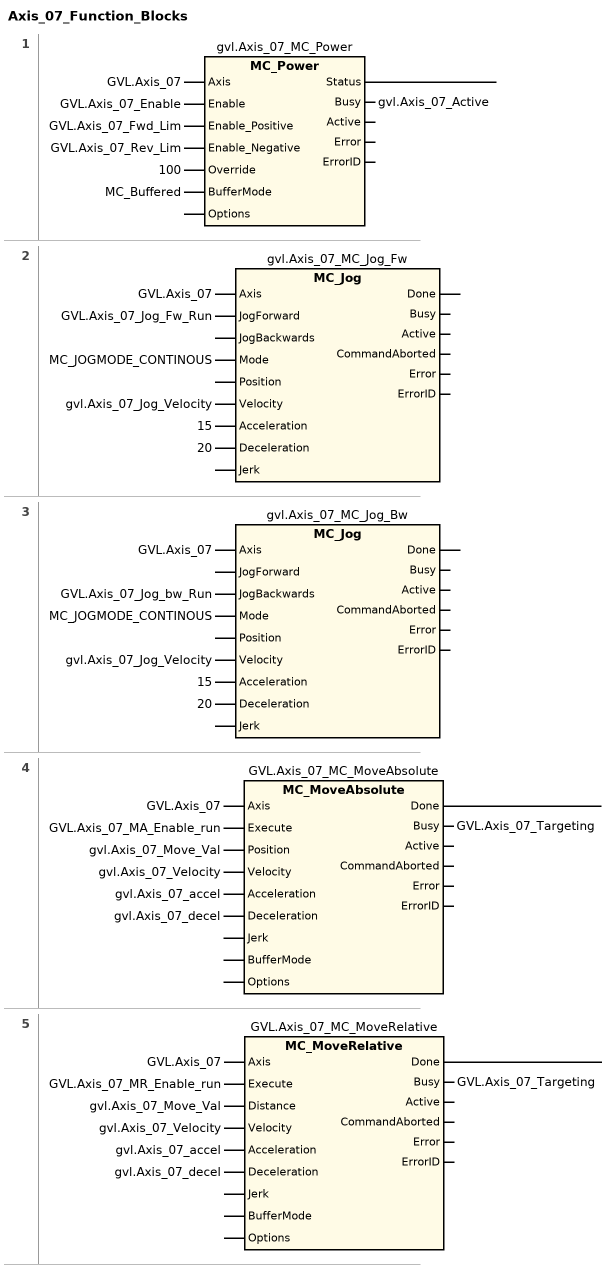
// NETWORK 1
gvl.Axis_07_MC_Power(
    Axis := GVL.Axis_07,
    Enable := GVL.Axis_07_Enable,
    Enable_Positive := GVL.Axis_07_Fwd_Lim,
    Enable_Negative := GVL.Axis_07_Rev_Lim,
    Override := 100,
    BufferMode := MC_Buffered,
    Busy => gvl.Axis_07_Active); // MC_Power

// NETWORK 2
gvl.Axis_07_MC_Jog_Fw(
    Axis := GVL.Axis_07,
    JogForward := GVL.Axis_07_Jog_Fw_Run,
    Mode := MC_JOGMODE_CONTINOUS,
    Velocity := gvl.Axis_07_Jog_Velocity,
    Acceleration := 15,
    Deceleration := 20); // MC_Jog

// NETWORK 3
gvl.Axis_07_MC_Jog_Bw(
    Axis := GVL.Axis_07,
    JogBackwards := GVL.Axis_07_Jog_bw_Run,
    Mode := MC_JOGMODE_CONTINOUS,
    Velocity := gvl.Axis_07_Jog_Velocity,
    Acceleration := 15,
    Deceleration := 20); // MC_Jog

// NETWORK 4
GVL.Axis_07_MC_MoveAbsolute(
    Axis := GVL.Axis_07,
    Execute := GVL.Axis_07_MA_Enable_run,
    Position := gvl.Axis_07_Move_Val,
    Velocity := gvl.Axis_07_Velocity,
    Acceleration := gvl.Axis_07_accel,
    Deceleration := gvl.Axis_07_decel,
    Busy => GVL.Axis_07_Targeting); // MC_MoveAbsolute

// NETWORK 5
GVL.Axis_07_MC_MoveRelative(
    Axis := GVL.Axis_07,
    Execute := GVL.Axis_07_MR_Enable_run,
    Distance := gvl.Axis_07_Move_Val,
    Velocity := gvl.Axis_07_Velocity,
    Acceleration := gvl.Axis_07_accel,
    Deceleration := gvl.Axis_07_decel,
    Busy => GVL.Axis_07_Targeting); // MC_MoveRelative

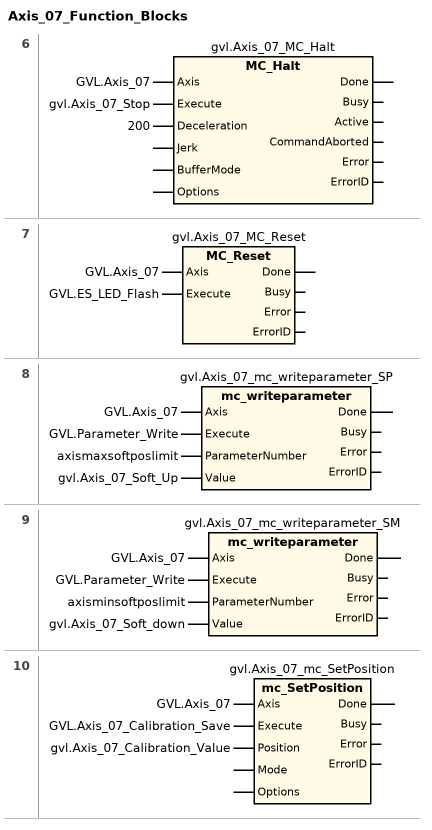
// NETWORK 6
gvl.Axis_07_MC_Halt(Axis := GVL.Axis_07, Execute := gvl.Axis_07_Stop, Deceleration := 200); // MC_Halt

// NETWORK 7
gvl.Axis_07_MC_Reset(Axis := GVL.Axis_07, Execute := GVL.ES_LED_Flash); // MC_Reset

// NETWORK 8
gvl.Axis_07_mc_writeparameter_SP(
    Axis := GVL.Axis_07,
    Execute := GVL.Parameter_Write,
    ParameterNumber := axismaxsoftposlimit,
    Value := gvl.Axis_07_Soft_Up); // mc_writeparameter

// NETWORK 9
gvl.Axis_07_mc_writeparameter_SM(
    Axis := GVL.Axis_07,
    Execute := GVL.Parameter_Write,
    ParameterNumber := axisminsoftposlimit,
    Value := gvl.Axis_07_Soft_down); // mc_writeparameter

// NETWORK 10
gvl.Axis_07_mc_SetPosition(
    Axis := GVL.Axis_07,
    Execute := GVL.Axis_07_Calibration_Save,
    Position := gvl.Axis_07_Calibration_Value); // mc_SetPosition

END_PROGRAM

// ---- POUs/Axis_07_Logic.TcPOU
PROGRAM Axis_07_Logic
VAR
	TON_0: TON;
	TON_1: TON;
	TON_2: TON;
	TON_3: TON;
	Axis_07_Velocity_Range: LREAL;
	Axis_07_Velocity_Scale: LREAL;
	Axis_07_Velocity_Raw: LREAL;
	Axis_07_Soft_Range: LREAL;
	Axis_07_Soft_Position: LREAL;
	Axis_07_Soft_Position_In_Range: LREAL;
END_VAR

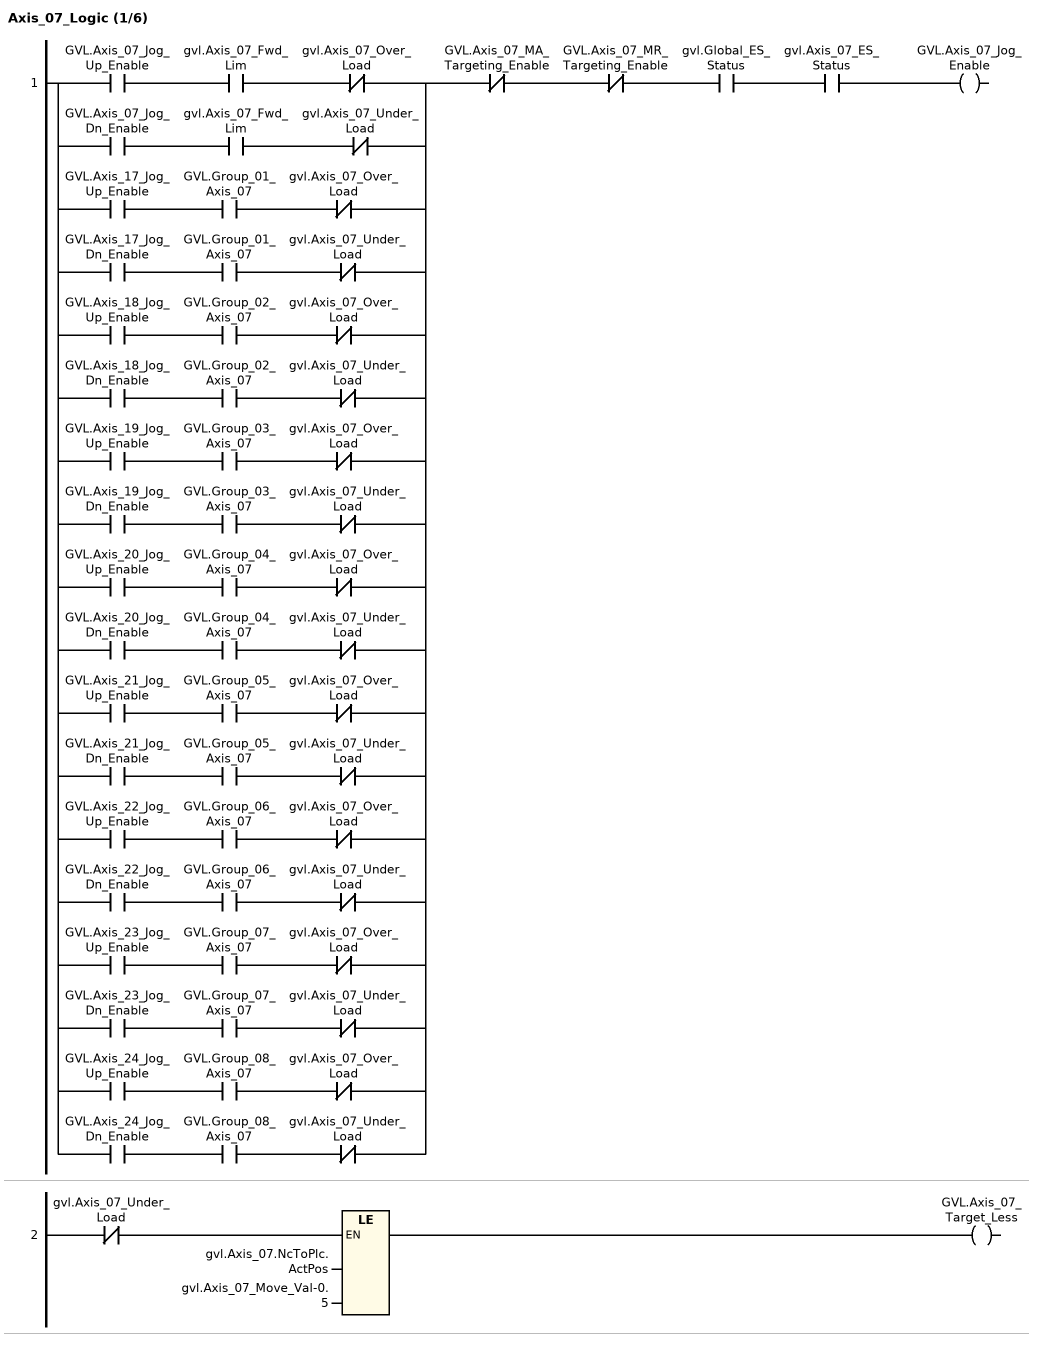
// NETWORK 1
GVL.Axis_07_Jog_Enable := (GVL.Axis_07_Jog_Up_Enable AND gvl.Axis_07_Fwd_Lim AND NOT gvl.Axis_07_Over_Load OR GVL.Axis_07_Jog_Dn_Enable AND gvl.Axis_07_Fwd_Lim AND NOT gvl.Axis_07_Under_Load OR GVL.Axis_17_Jog_Up_Enable AND GVL.Group_01_Axis_07 AND NOT gvl.Axis_07_Over_Load OR GVL.Axis_17_Jog_Dn_Enable AND GVL.Group_01_Axis_07 AND NOT gvl.Axis_07_Under_Load OR GVL.Axis_18_Jog_Up_Enable AND GVL.Group_02_Axis_07 AND NOT gvl.Axis_07_Over_Load OR GVL.Axis_18_Jog_Dn_Enable AND GVL.Group_02_Axis_07 AND NOT gvl.Axis_07_Under_Load OR GVL.Axis_19_Jog_Up_Enable AND GVL.Group_03_Axis_07 AND NOT gvl.Axis_07_Over_Load OR GVL.Axis_19_Jog_Dn_Enable AND GVL.Group_03_Axis_07 AND NOT gvl.Axis_07_Under_Load OR GVL.Axis_20_Jog_Up_Enable AND GVL.Group_04_Axis_07 AND NOT gvl.Axis_07_Over_Load OR GVL.Axis_20_Jog_Dn_Enable AND GVL.Group_04_Axis_07 AND NOT gvl.Axis_07_Under_Load OR GVL.Axis_21_Jog_Up_Enable AND GVL.Group_05_Axis_07 AND NOT gvl.Axis_07_Over_Load OR GVL.Axis_21_Jog_Dn_Enable AND GVL.Group_05_Axis_07 AND NOT gvl.Axis_07_Under_Load OR GVL.Axis_22_Jog_Up_Enable AND GVL.Group_06_Axis_07 AND NOT gvl.Axis_07_Over_Load OR GVL.Axis_22_Jog_Dn_Enable AND GVL.Group_06_Axis_07 AND NOT gvl.Axis_07_Under_Load OR GVL.Axis_23_Jog_Up_Enable AND GVL.Group_07_Axis_07 AND NOT gvl.Axis_07_Over_Load OR GVL.Axis_23_Jog_Dn_Enable AND GVL.Group_07_Axis_07 AND NOT gvl.Axis_07_Under_Load OR GVL.Axis_24_Jog_Up_Enable AND GVL.Group_08_Axis_07 AND NOT gvl.Axis_07_Over_Load OR GVL.Axis_24_Jog_Dn_Enable AND GVL.Group_08_Axis_07 AND NOT gvl.Axis_07_Under_Load) AND NOT GVL.Axis_07_MA_Targeting_Enable AND NOT GVL.Axis_07_MR_Targeting_Enable AND gvl.Global_ES_Status AND gvl.Axis_07_ES_Status;

// NETWORK 2
GVL.Axis_07_Target_Less := NOT gvl.Axis_07_Under_Load AND gvl.Axis_07.NcToPlc.ActPos <= (gvl.Axis_07_Move_Val-0.5);

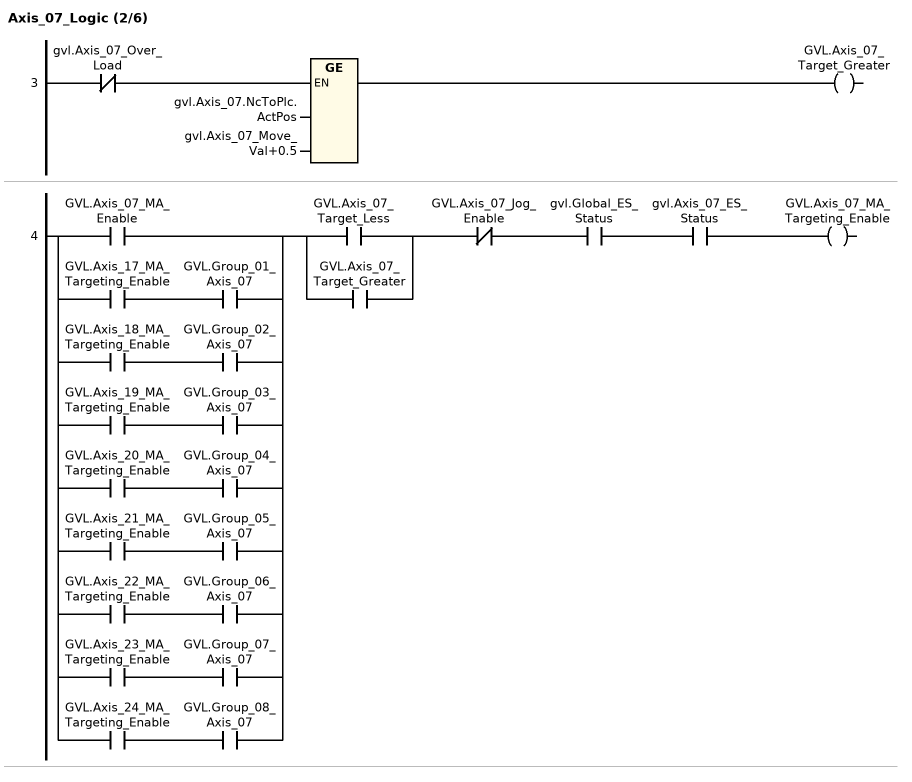
// NETWORK 3
GVL.Axis_07_Target_Greater := NOT gvl.Axis_07_Over_Load AND gvl.Axis_07.NcToPlc.ActPos >= (gvl.Axis_07_Move_Val+0.5);

// NETWORK 4
GVL.Axis_07_MA_Targeting_Enable := (GVL.Axis_07_MA_Enable OR GVL.Axis_17_MA_Targeting_Enable AND GVL.Group_01_Axis_07 OR GVL.Axis_18_MA_Targeting_Enable AND GVL.Group_02_Axis_07 OR GVL.Axis_19_MA_Targeting_Enable AND GVL.Group_03_Axis_07 OR GVL.Axis_20_MA_Targeting_Enable AND GVL.Group_04_Axis_07 OR GVL.Axis_21_MA_Targeting_Enable AND GVL.Group_05_Axis_07 OR GVL.Axis_22_MA_Targeting_Enable AND GVL.Group_06_Axis_07 OR GVL.Axis_23_MA_Targeting_Enable AND GVL.Group_07_Axis_07 OR GVL.Axis_24_MA_Targeting_Enable AND GVL.Group_08_Axis_07) AND (GVL.Axis_07_Target_Less OR GVL.Axis_07_Target_Greater) AND NOT GVL.Axis_07_Jog_Enable AND gvl.Global_ES_Status AND gvl.Axis_07_ES_Status;

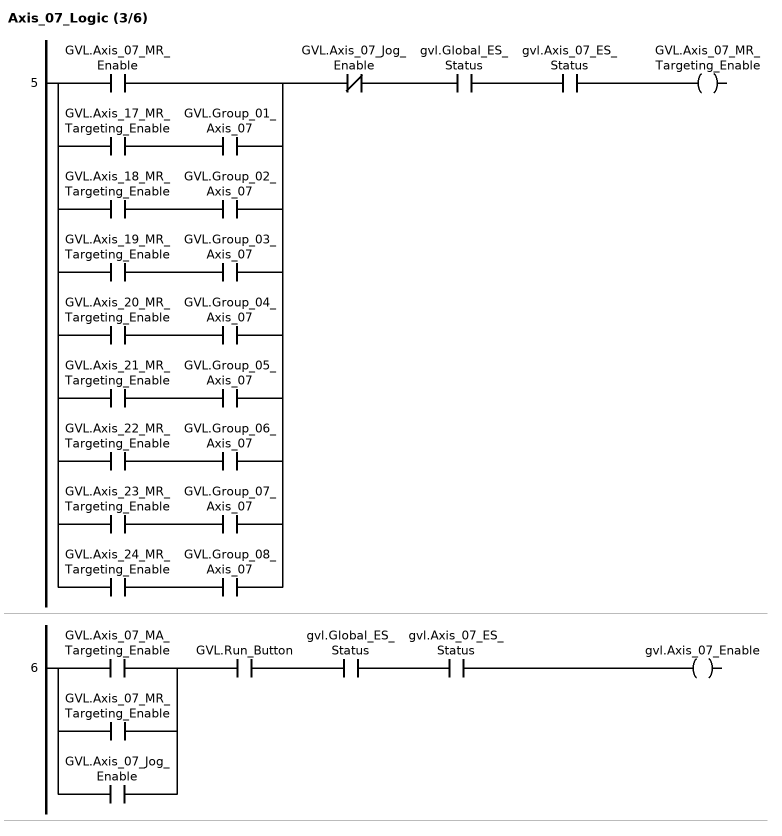
// NETWORK 5
GVL.Axis_07_MR_Targeting_Enable := (GVL.Axis_07_MR_Enable OR GVL.Axis_17_MR_Targeting_Enable AND GVL.Group_01_Axis_07 OR GVL.Axis_18_MR_Targeting_Enable AND GVL.Group_02_Axis_07 OR GVL.Axis_19_MR_Targeting_Enable AND GVL.Group_03_Axis_07 OR GVL.Axis_20_MR_Targeting_Enable AND GVL.Group_04_Axis_07 OR GVL.Axis_21_MR_Targeting_Enable AND GVL.Group_05_Axis_07 OR GVL.Axis_22_MR_Targeting_Enable AND GVL.Group_06_Axis_07 OR GVL.Axis_23_MR_Targeting_Enable AND GVL.Group_07_Axis_07 OR GVL.Axis_24_MR_Targeting_Enable AND GVL.Group_08_Axis_07) AND NOT GVL.Axis_07_Jog_Enable AND gvl.Global_ES_Status AND gvl.Axis_07_ES_Status;

// NETWORK 6
gvl.Axis_07_Enable := (GVL.Axis_07_MA_Targeting_Enable OR GVL.Axis_07_MR_Targeting_Enable OR GVL.Axis_07_Jog_Enable) AND GVL.Run_Button AND gvl.Global_ES_Status AND gvl.Axis_07_ES_Status;

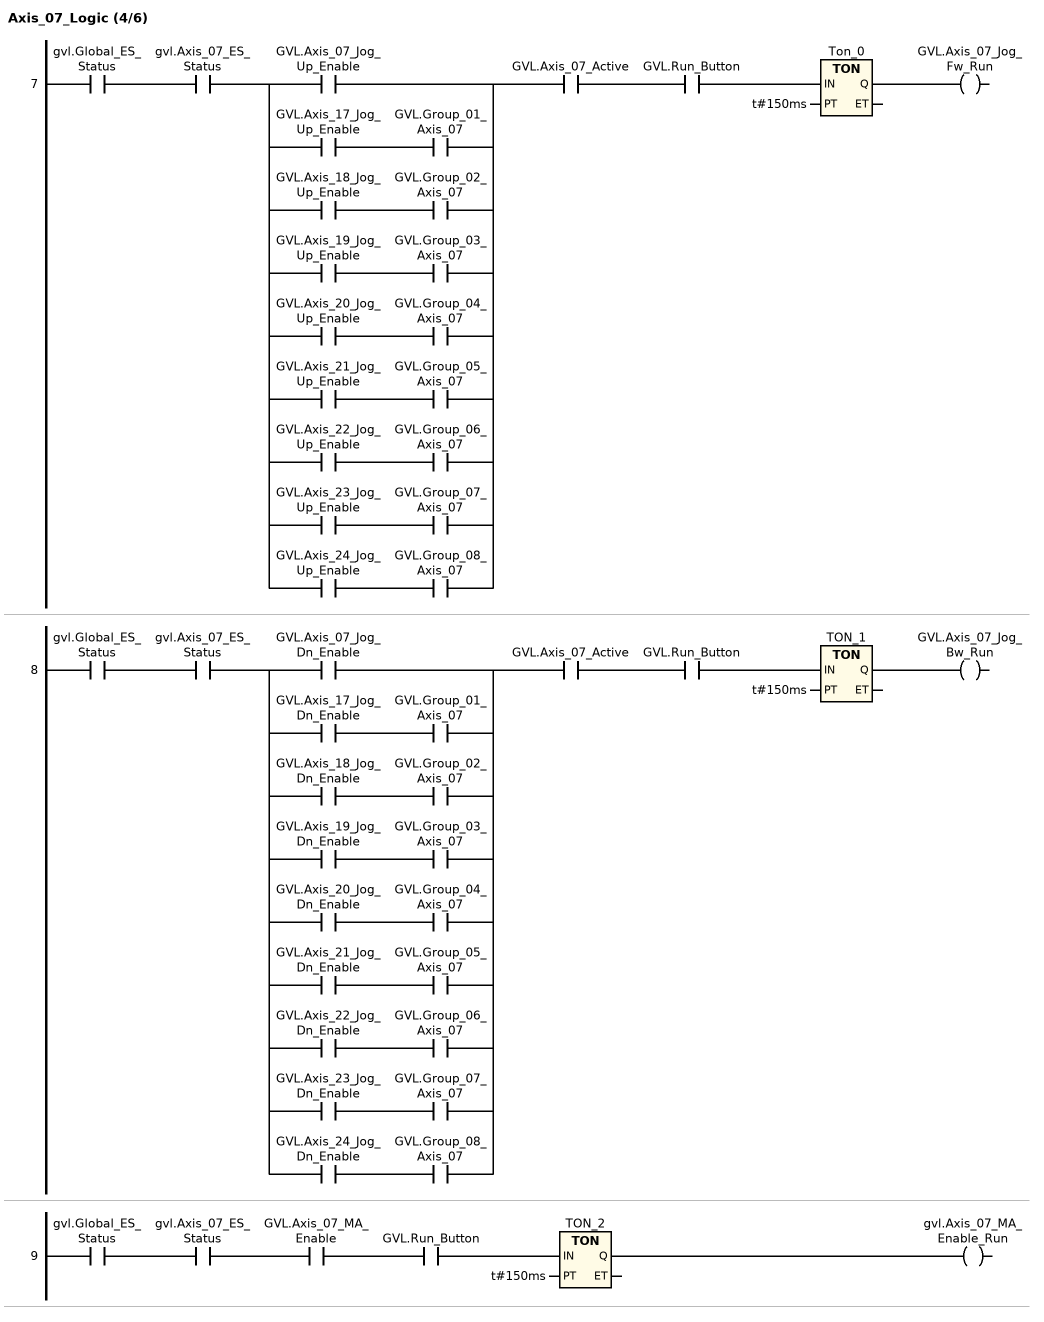
// NETWORK 7
Ton_0(IN := gvl.Global_ES_Status AND gvl.Axis_07_ES_Status AND (GVL.Axis_07_Jog_Up_Enable OR GVL.Axis_17_Jog_Up_Enable AND GVL.Group_01_Axis_07 OR GVL.Axis_18_Jog_Up_Enable AND GVL.Group_02_Axis_07 OR GVL.Axis_19_Jog_Up_Enable AND GVL.Group_03_Axis_07 OR GVL.Axis_20_Jog_Up_Enable AND GVL.Group_04_Axis_07 OR GVL.Axis_21_Jog_Up_Enable AND GVL.Group_05_Axis_07 OR GVL.Axis_22_Jog_Up_Enable AND GVL.Group_06_Axis_07 OR GVL.Axis_23_Jog_Up_Enable AND GVL.Group_07_Axis_07 OR GVL.Axis_24_Jog_Up_Enable AND GVL.Group_08_Axis_07) AND GVL.Axis_07_Active AND GVL.Run_Button, PT := t#150ms); // TON
GVL.Axis_07_Jog_Fw_Run := Ton_0.Q;

// NETWORK 8
TON_1(IN := gvl.Global_ES_Status AND gvl.Axis_07_ES_Status AND (GVL.Axis_07_Jog_Dn_Enable OR GVL.Axis_17_Jog_Dn_Enable AND GVL.Group_01_Axis_07 OR GVL.Axis_18_Jog_Dn_Enable AND GVL.Group_02_Axis_07 OR GVL.Axis_19_Jog_Dn_Enable AND GVL.Group_03_Axis_07 OR GVL.Axis_20_Jog_Dn_Enable AND GVL.Group_04_Axis_07 OR GVL.Axis_21_Jog_Dn_Enable AND GVL.Group_05_Axis_07 OR GVL.Axis_22_Jog_Dn_Enable AND GVL.Group_06_Axis_07 OR GVL.Axis_23_Jog_Dn_Enable AND GVL.Group_07_Axis_07 OR GVL.Axis_24_Jog_Dn_Enable AND GVL.Group_08_Axis_07) AND GVL.Axis_07_Active AND GVL.Run_Button, PT := t#150ms); // TON
GVL.Axis_07_Jog_Bw_Run := TON_1.Q;

// NETWORK 9
TON_2(IN := gvl.Global_ES_Status AND gvl.Axis_07_ES_Status AND GVL.Axis_07_MA_Enable AND GVL.Run_Button, PT := t#150ms); // TON
gvl.Axis_07_MA_Enable_Run := TON_2.Q;

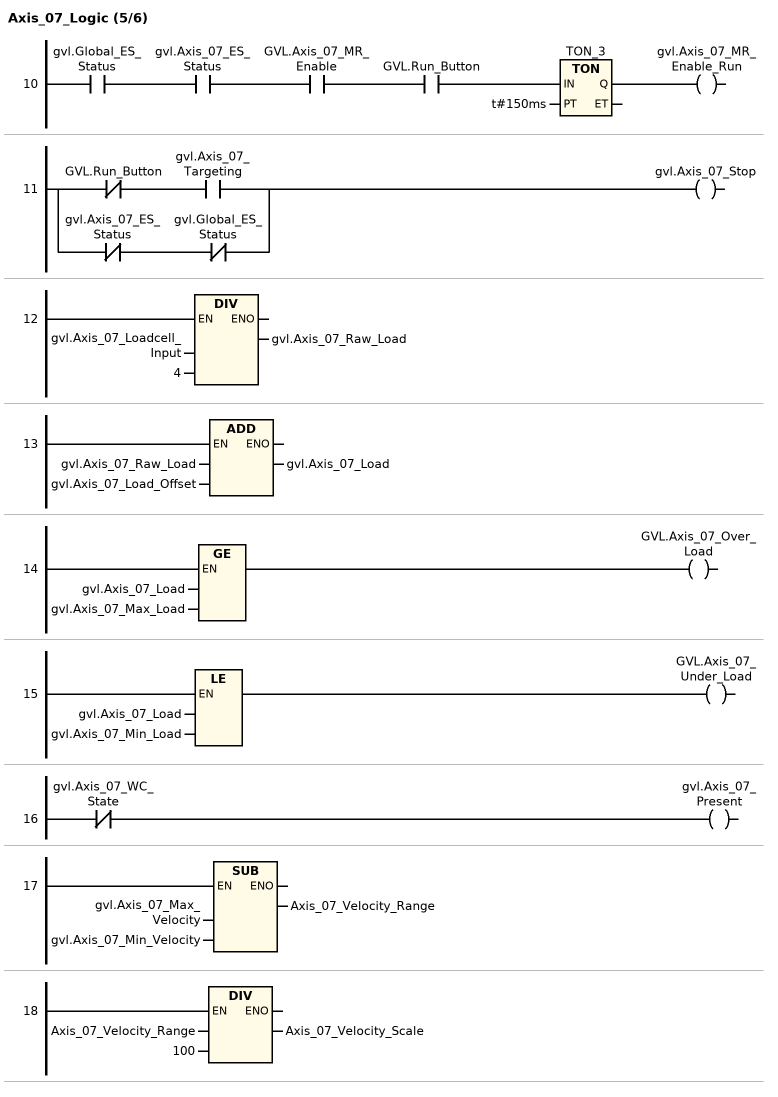
// NETWORK 10
TON_3(IN := gvl.Global_ES_Status AND gvl.Axis_07_ES_Status AND GVL.Axis_07_MR_Enable AND GVL.Run_Button, PT := t#150ms); // TON
gvl.Axis_07_MR_Enable_Run := TON_3.Q;

// NETWORK 11
gvl.Axis_07_Stop := NOT GVL.Run_Button AND gvl.Axis_07_Targeting OR NOT gvl.Axis_07_ES_Status AND NOT gvl.Global_ES_Status;

// NETWORK 12
gvl.Axis_07_Raw_Load := gvl.Axis_07_Loadcell_Input / 4;

// NETWORK 13
gvl.Axis_07_Load := gvl.Axis_07_Raw_Load + gvl.Axis_07_Load_Offset;

// NETWORK 14
GVL.Axis_07_Over_Load := gvl.Axis_07_Load >= gvl.Axis_07_Max_Load;

// NETWORK 15
GVL.Axis_07_Under_Load := gvl.Axis_07_Load <= gvl.Axis_07_Min_Load;

// NETWORK 16
gvl.Axis_07_Present := NOT gvl.Axis_07_WC_State;

// NETWORK 17
Axis_07_Velocity_Range := gvl.Axis_07_Max_Velocity - gvl.Axis_07_Min_Velocity;

// NETWORK 18
Axis_07_Velocity_Scale := Axis_07_Velocity_Range / 100;

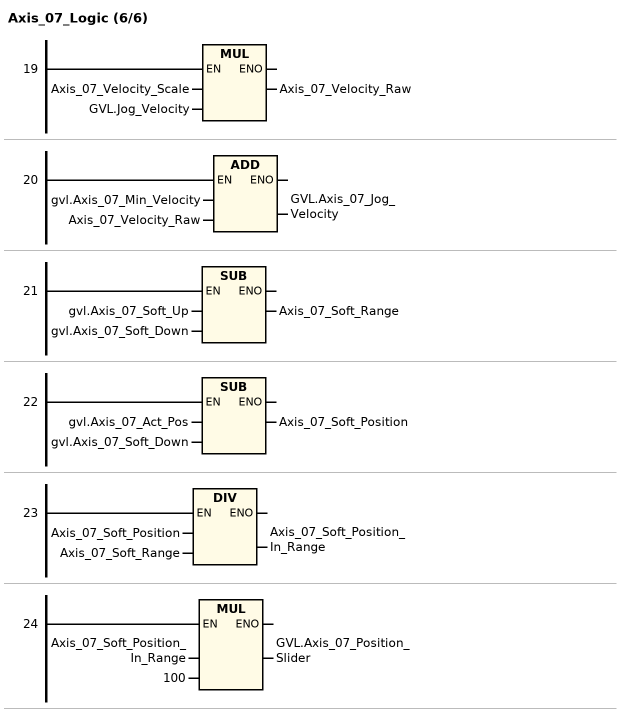
// NETWORK 19
Axis_07_Velocity_Raw := Axis_07_Velocity_Scale * GVL.Jog_Velocity;

// NETWORK 20
GVL.Axis_07_Jog_Velocity := gvl.Axis_07_Min_Velocity + Axis_07_Velocity_Raw;

// NETWORK 21
Axis_07_Soft_Range := gvl.Axis_07_Soft_Up - gvl.Axis_07_Soft_Down;

// NETWORK 22
Axis_07_Soft_Position := gvl.Axis_07_Act_Pos - gvl.Axis_07_Soft_Down;

// NETWORK 23
Axis_07_Soft_Position_In_Range := Axis_07_Soft_Position / Axis_07_Soft_Range;

// NETWORK 24
GVL.Axis_07_Position_Slider := Axis_07_Soft_Position_In_Range * 100;

END_PROGRAM

// ---- POUs/Axis_08_Function_Blocks.TcPOU
PROGRAM Axis_08_Function_Blocks
VAR
END_VAR

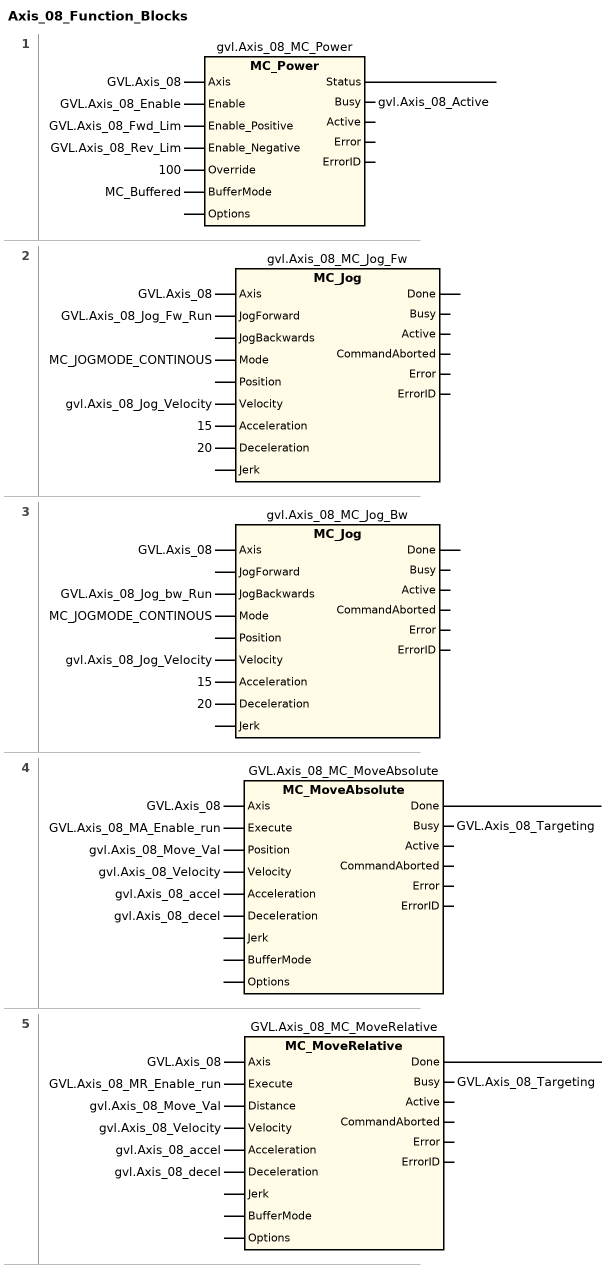
// NETWORK 1
gvl.Axis_08_MC_Power(
    Axis := GVL.Axis_08,
    Enable := GVL.Axis_08_Enable,
    Enable_Positive := GVL.Axis_08_Fwd_Lim,
    Enable_Negative := GVL.Axis_08_Rev_Lim,
    Override := 100,
    BufferMode := MC_Buffered,
    Busy => gvl.Axis_08_Active); // MC_Power

// NETWORK 2
gvl.Axis_08_MC_Jog_Fw(
    Axis := GVL.Axis_08,
    JogForward := GVL.Axis_08_Jog_Fw_Run,
    Mode := MC_JOGMODE_CONTINOUS,
    Velocity := gvl.Axis_08_Jog_Velocity,
    Acceleration := 15,
    Deceleration := 20); // MC_Jog

// NETWORK 3
gvl.Axis_08_MC_Jog_Bw(
    Axis := GVL.Axis_08,
    JogBackwards := GVL.Axis_08_Jog_bw_Run,
    Mode := MC_JOGMODE_CONTINOUS,
    Velocity := gvl.Axis_08_Jog_Velocity,
    Acceleration := 15,
    Deceleration := 20); // MC_Jog

// NETWORK 4
GVL.Axis_08_MC_MoveAbsolute(
    Axis := GVL.Axis_08,
    Execute := GVL.Axis_08_MA_Enable_run,
    Position := gvl.Axis_08_Move_Val,
    Velocity := gvl.Axis_08_Velocity,
    Acceleration := gvl.Axis_08_accel,
    Deceleration := gvl.Axis_08_decel,
    Busy => GVL.Axis_08_Targeting); // MC_MoveAbsolute

// NETWORK 5
GVL.Axis_08_MC_MoveRelative(
    Axis := GVL.Axis_08,
    Execute := GVL.Axis_08_MR_Enable_run,
    Distance := gvl.Axis_08_Move_Val,
    Velocity := gvl.Axis_08_Velocity,
    Acceleration := gvl.Axis_08_accel,
    Deceleration := gvl.Axis_08_decel,
    Busy => GVL.Axis_08_Targeting); // MC_MoveRelative

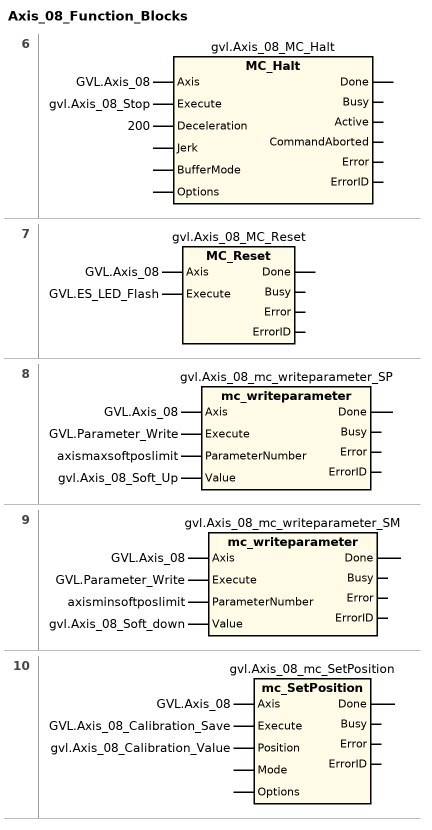
// NETWORK 6
gvl.Axis_08_MC_Halt(Axis := GVL.Axis_08, Execute := gvl.Axis_08_Stop, Deceleration := 200); // MC_Halt

// NETWORK 7
gvl.Axis_08_MC_Reset(Axis := GVL.Axis_08, Execute := GVL.ES_LED_Flash); // MC_Reset

// NETWORK 8
gvl.Axis_08_mc_writeparameter_SP(
    Axis := GVL.Axis_08,
    Execute := GVL.Parameter_Write,
    ParameterNumber := axismaxsoftposlimit,
    Value := gvl.Axis_08_Soft_Up); // mc_writeparameter

// NETWORK 9
gvl.Axis_08_mc_writeparameter_SM(
    Axis := GVL.Axis_08,
    Execute := GVL.Parameter_Write,
    ParameterNumber := axisminsoftposlimit,
    Value := gvl.Axis_08_Soft_down); // mc_writeparameter

// NETWORK 10
gvl.Axis_08_mc_SetPosition(
    Axis := GVL.Axis_08,
    Execute := GVL.Axis_08_Calibration_Save,
    Position := gvl.Axis_08_Calibration_Value); // mc_SetPosition

END_PROGRAM

// ---- POUs/Axis_08_Logic.TcPOU
PROGRAM Axis_08_Logic
VAR
	TON_0: TON;
	TON_1: TON;
	TON_2: TON;
	TON_3: TON;
	Axis_08_Velocity_Range: LREAL;
	Axis_08_Velocity_Scale: LREAL;
	Axis_08_Velocity_Raw: LREAL;
	Axis_08_Soft_Range: LREAL;
	Axis_08_Soft_Position: LREAL;
	Axis_08_Soft_Position_In_Range: LREAL;
END_VAR

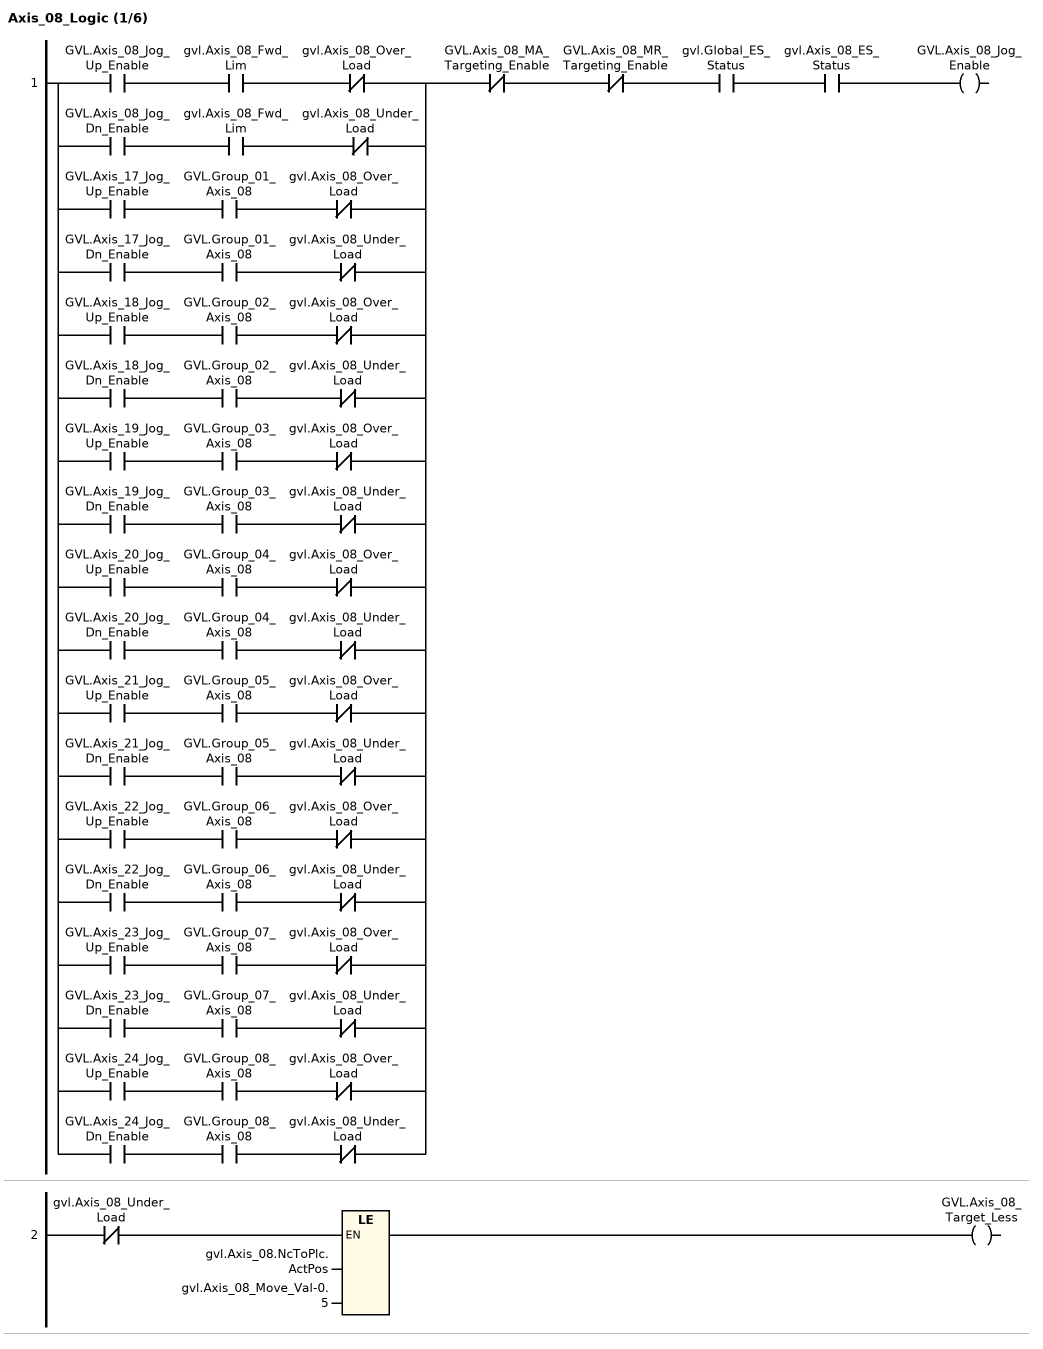
// NETWORK 1
GVL.Axis_08_Jog_Enable := (GVL.Axis_08_Jog_Up_Enable AND gvl.Axis_08_Fwd_Lim AND NOT gvl.Axis_08_Over_Load OR GVL.Axis_08_Jog_Dn_Enable AND gvl.Axis_08_Fwd_Lim AND NOT gvl.Axis_08_Under_Load OR GVL.Axis_17_Jog_Up_Enable AND GVL.Group_01_Axis_08 AND NOT gvl.Axis_08_Over_Load OR GVL.Axis_17_Jog_Dn_Enable AND GVL.Group_01_Axis_08 AND NOT gvl.Axis_08_Under_Load OR GVL.Axis_18_Jog_Up_Enable AND GVL.Group_02_Axis_08 AND NOT gvl.Axis_08_Over_Load OR GVL.Axis_18_Jog_Dn_Enable AND GVL.Group_02_Axis_08 AND NOT gvl.Axis_08_Under_Load OR GVL.Axis_19_Jog_Up_Enable AND GVL.Group_03_Axis_08 AND NOT gvl.Axis_08_Over_Load OR GVL.Axis_19_Jog_Dn_Enable AND GVL.Group_03_Axis_08 AND NOT gvl.Axis_08_Under_Load OR GVL.Axis_20_Jog_Up_Enable AND GVL.Group_04_Axis_08 AND NOT gvl.Axis_08_Over_Load OR GVL.Axis_20_Jog_Dn_Enable AND GVL.Group_04_Axis_08 AND NOT gvl.Axis_08_Under_Load OR GVL.Axis_21_Jog_Up_Enable AND GVL.Group_05_Axis_08 AND NOT gvl.Axis_08_Over_Load OR GVL.Axis_21_Jog_Dn_Enable AND GVL.Group_05_Axis_08 AND NOT gvl.Axis_08_Under_Load OR GVL.Axis_22_Jog_Up_Enable AND GVL.Group_06_Axis_08 AND NOT gvl.Axis_08_Over_Load OR GVL.Axis_22_Jog_Dn_Enable AND GVL.Group_06_Axis_08 AND NOT gvl.Axis_08_Under_Load OR GVL.Axis_23_Jog_Up_Enable AND GVL.Group_07_Axis_08 AND NOT gvl.Axis_08_Over_Load OR GVL.Axis_23_Jog_Dn_Enable AND GVL.Group_07_Axis_08 AND NOT gvl.Axis_08_Under_Load OR GVL.Axis_24_Jog_Up_Enable AND GVL.Group_08_Axis_08 AND NOT gvl.Axis_08_Over_Load OR GVL.Axis_24_Jog_Dn_Enable AND GVL.Group_08_Axis_08 AND NOT gvl.Axis_08_Under_Load) AND NOT GVL.Axis_08_MA_Targeting_Enable AND NOT GVL.Axis_08_MR_Targeting_Enable AND gvl.Global_ES_Status AND gvl.Axis_08_ES_Status;

// NETWORK 2
GVL.Axis_08_Target_Less := NOT gvl.Axis_08_Under_Load AND gvl.Axis_08.NcToPlc.ActPos <= (gvl.Axis_08_Move_Val-0.5);

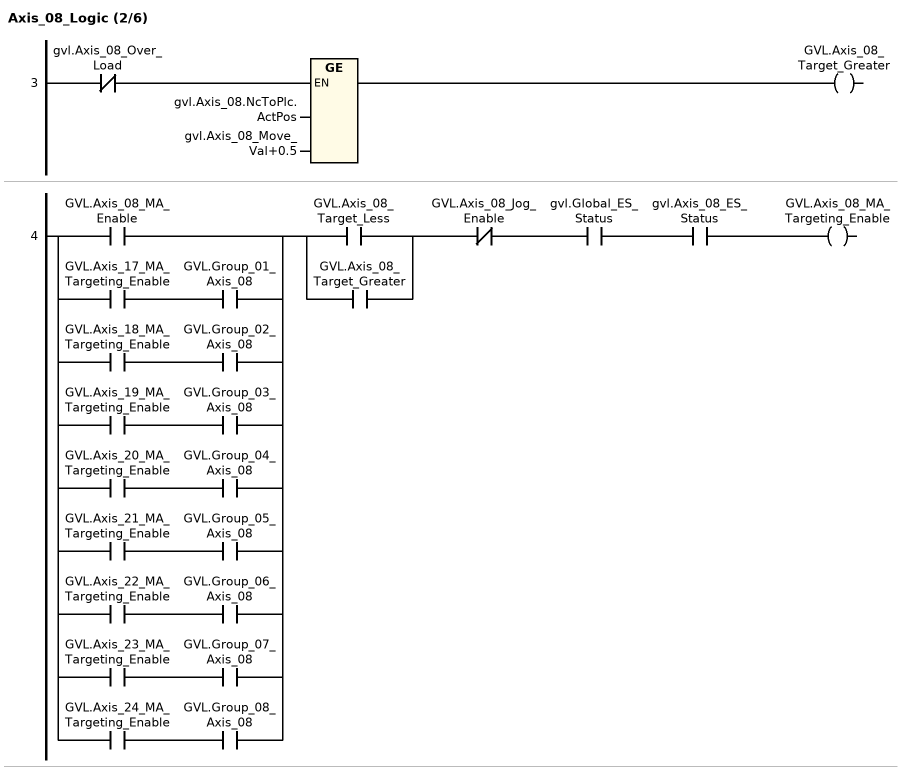
// NETWORK 3
GVL.Axis_08_Target_Greater := NOT gvl.Axis_08_Over_Load AND gvl.Axis_08.NcToPlc.ActPos >= (gvl.Axis_08_Move_Val+0.5);

// NETWORK 4
GVL.Axis_08_MA_Targeting_Enable := (GVL.Axis_08_MA_Enable OR GVL.Axis_17_MA_Targeting_Enable AND GVL.Group_01_Axis_08 OR GVL.Axis_18_MA_Targeting_Enable AND GVL.Group_02_Axis_08 OR GVL.Axis_19_MA_Targeting_Enable AND GVL.Group_03_Axis_08 OR GVL.Axis_20_MA_Targeting_Enable AND GVL.Group_04_Axis_08 OR GVL.Axis_21_MA_Targeting_Enable AND GVL.Group_05_Axis_08 OR GVL.Axis_22_MA_Targeting_Enable AND GVL.Group_06_Axis_08 OR GVL.Axis_23_MA_Targeting_Enable AND GVL.Group_07_Axis_08 OR GVL.Axis_24_MA_Targeting_Enable AND GVL.Group_08_Axis_08) AND (GVL.Axis_08_Target_Less OR GVL.Axis_08_Target_Greater) AND NOT GVL.Axis_08_Jog_Enable AND gvl.Global_ES_Status AND gvl.Axis_08_ES_Status;

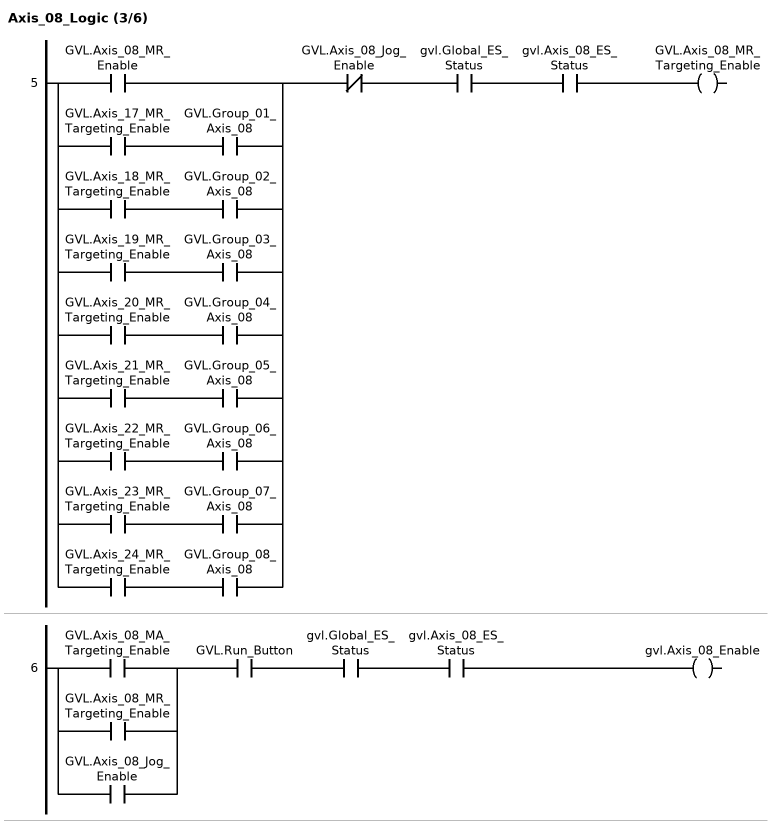
// NETWORK 5
GVL.Axis_08_MR_Targeting_Enable := (GVL.Axis_08_MR_Enable OR GVL.Axis_17_MR_Targeting_Enable AND GVL.Group_01_Axis_08 OR GVL.Axis_18_MR_Targeting_Enable AND GVL.Group_02_Axis_08 OR GVL.Axis_19_MR_Targeting_Enable AND GVL.Group_03_Axis_08 OR GVL.Axis_20_MR_Targeting_Enable AND GVL.Group_04_Axis_08 OR GVL.Axis_21_MR_Targeting_Enable AND GVL.Group_05_Axis_08 OR GVL.Axis_22_MR_Targeting_Enable AND GVL.Group_06_Axis_08 OR GVL.Axis_23_MR_Targeting_Enable AND GVL.Group_07_Axis_08 OR GVL.Axis_24_MR_Targeting_Enable AND GVL.Group_08_Axis_08) AND NOT GVL.Axis_08_Jog_Enable AND gvl.Global_ES_Status AND gvl.Axis_08_ES_Status;

// NETWORK 6
gvl.Axis_08_Enable := (GVL.Axis_08_MA_Targeting_Enable OR GVL.Axis_08_MR_Targeting_Enable OR GVL.Axis_08_Jog_Enable) AND GVL.Run_Button AND gvl.Global_ES_Status AND gvl.Axis_08_ES_Status;

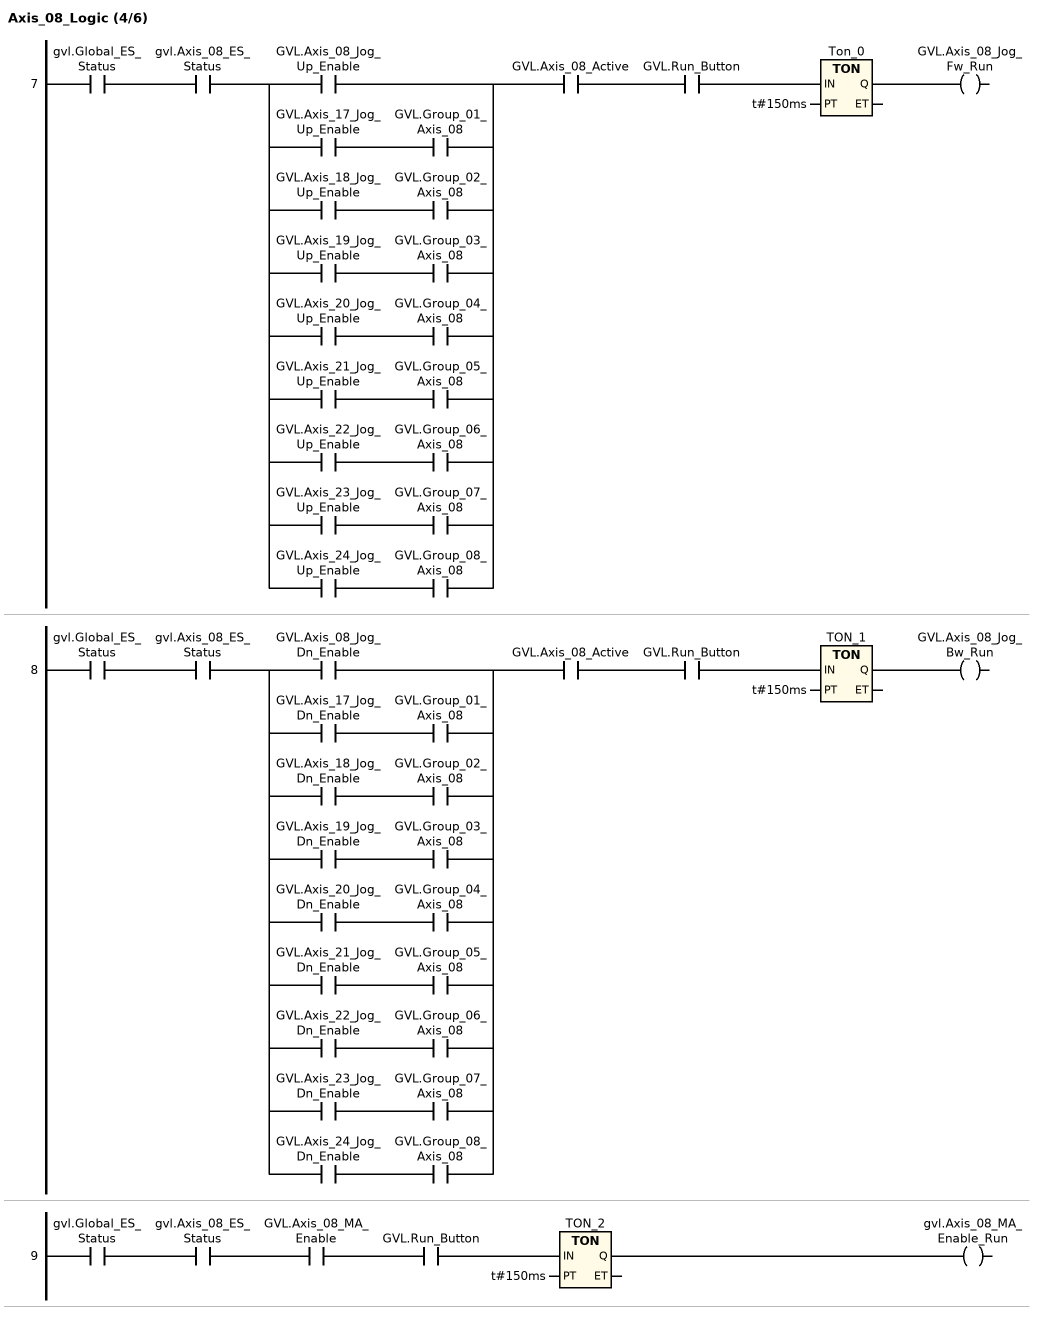
// NETWORK 7
Ton_0(IN := gvl.Global_ES_Status AND gvl.Axis_08_ES_Status AND (GVL.Axis_08_Jog_Up_Enable OR GVL.Axis_17_Jog_Up_Enable AND GVL.Group_01_Axis_08 OR GVL.Axis_18_Jog_Up_Enable AND GVL.Group_02_Axis_08 OR GVL.Axis_19_Jog_Up_Enable AND GVL.Group_03_Axis_08 OR GVL.Axis_20_Jog_Up_Enable AND GVL.Group_04_Axis_08 OR GVL.Axis_21_Jog_Up_Enable AND GVL.Group_05_Axis_08 OR GVL.Axis_22_Jog_Up_Enable AND GVL.Group_06_Axis_08 OR GVL.Axis_23_Jog_Up_Enable AND GVL.Group_07_Axis_08 OR GVL.Axis_24_Jog_Up_Enable AND GVL.Group_08_Axis_08) AND GVL.Axis_08_Active AND GVL.Run_Button, PT := t#150ms); // TON
GVL.Axis_08_Jog_Fw_Run := Ton_0.Q;

// NETWORK 8
TON_1(IN := gvl.Global_ES_Status AND gvl.Axis_08_ES_Status AND (GVL.Axis_08_Jog_Dn_Enable OR GVL.Axis_17_Jog_Dn_Enable AND GVL.Group_01_Axis_08 OR GVL.Axis_18_Jog_Dn_Enable AND GVL.Group_02_Axis_08 OR GVL.Axis_19_Jog_Dn_Enable AND GVL.Group_03_Axis_08 OR GVL.Axis_20_Jog_Dn_Enable AND GVL.Group_04_Axis_08 OR GVL.Axis_21_Jog_Dn_Enable AND GVL.Group_05_Axis_08 OR GVL.Axis_22_Jog_Dn_Enable AND GVL.Group_06_Axis_08 OR GVL.Axis_23_Jog_Dn_Enable AND GVL.Group_07_Axis_08 OR GVL.Axis_24_Jog_Dn_Enable AND GVL.Group_08_Axis_08) AND GVL.Axis_08_Active AND GVL.Run_Button, PT := t#150ms); // TON
GVL.Axis_08_Jog_Bw_Run := TON_1.Q;

// NETWORK 9
TON_2(IN := gvl.Global_ES_Status AND gvl.Axis_08_ES_Status AND GVL.Axis_08_MA_Enable AND GVL.Run_Button, PT := t#150ms); // TON
gvl.Axis_08_MA_Enable_Run := TON_2.Q;

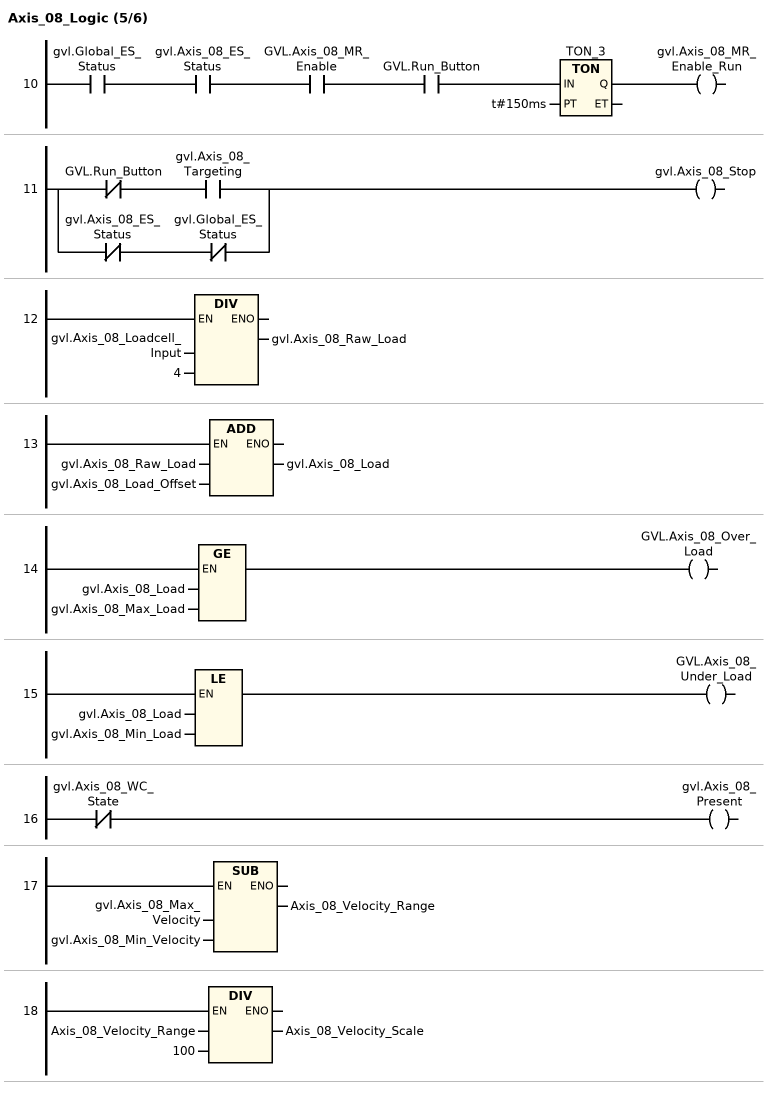
// NETWORK 10
TON_3(IN := gvl.Global_ES_Status AND gvl.Axis_08_ES_Status AND GVL.Axis_08_MR_Enable AND GVL.Run_Button, PT := t#150ms); // TON
gvl.Axis_08_MR_Enable_Run := TON_3.Q;

// NETWORK 11
gvl.Axis_08_Stop := NOT GVL.Run_Button AND gvl.Axis_08_Targeting OR NOT gvl.Axis_08_ES_Status AND NOT gvl.Global_ES_Status;

// NETWORK 12
gvl.Axis_08_Raw_Load := gvl.Axis_08_Loadcell_Input / 4;

// NETWORK 13
gvl.Axis_08_Load := gvl.Axis_08_Raw_Load + gvl.Axis_08_Load_Offset;

// NETWORK 14
GVL.Axis_08_Over_Load := gvl.Axis_08_Load >= gvl.Axis_08_Max_Load;

// NETWORK 15
GVL.Axis_08_Under_Load := gvl.Axis_08_Load <= gvl.Axis_08_Min_Load;

// NETWORK 16
gvl.Axis_08_Present := NOT gvl.Axis_08_WC_State;

// NETWORK 17
Axis_08_Velocity_Range := gvl.Axis_08_Max_Velocity - gvl.Axis_08_Min_Velocity;

// NETWORK 18
Axis_08_Velocity_Scale := Axis_08_Velocity_Range / 100;

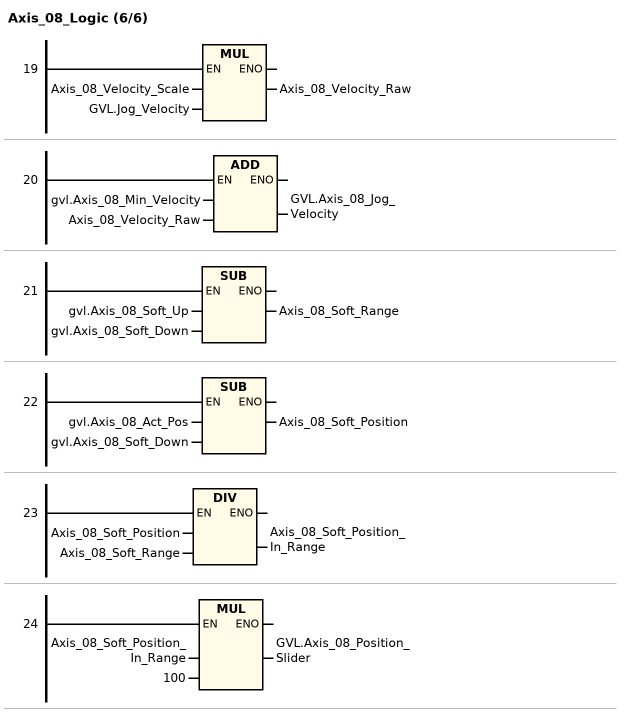
// NETWORK 19
Axis_08_Velocity_Raw := Axis_08_Velocity_Scale * GVL.Jog_Velocity;

// NETWORK 20
GVL.Axis_08_Jog_Velocity := gvl.Axis_08_Min_Velocity + Axis_08_Velocity_Raw;

// NETWORK 21
Axis_08_Soft_Range := gvl.Axis_08_Soft_Up - gvl.Axis_08_Soft_Down;

// NETWORK 22
Axis_08_Soft_Position := gvl.Axis_08_Act_Pos - gvl.Axis_08_Soft_Down;

// NETWORK 23
Axis_08_Soft_Position_In_Range := Axis_08_Soft_Position / Axis_08_Soft_Range;

// NETWORK 24
GVL.Axis_08_Position_Slider := Axis_08_Soft_Position_In_Range * 100;

END_PROGRAM

// ---- POUs/Axis_09_Function_Blocks.TcPOU
PROGRAM Axis_09_Function_Blocks
VAR
END_VAR

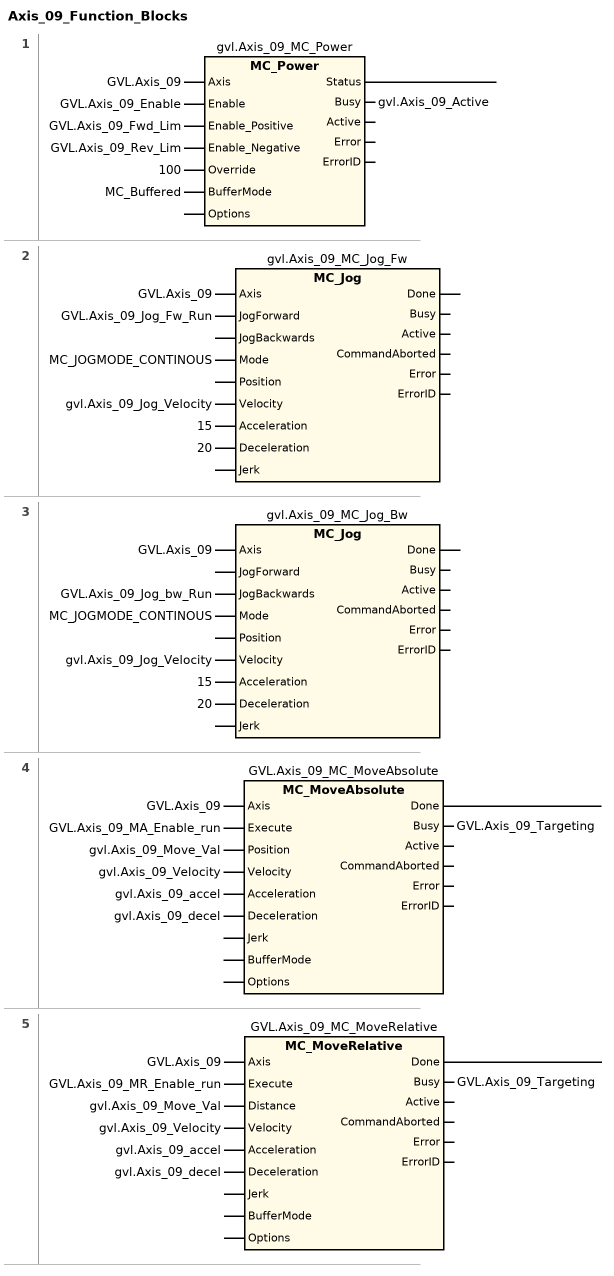
// NETWORK 1
gvl.Axis_09_MC_Power(
    Axis := GVL.Axis_09,
    Enable := GVL.Axis_09_Enable,
    Enable_Positive := GVL.Axis_09_Fwd_Lim,
    Enable_Negative := GVL.Axis_09_Rev_Lim,
    Override := 100,
    BufferMode := MC_Buffered,
    Busy => gvl.Axis_09_Active); // MC_Power

// NETWORK 2
gvl.Axis_09_MC_Jog_Fw(
    Axis := GVL.Axis_09,
    JogForward := GVL.Axis_09_Jog_Fw_Run,
    Mode := MC_JOGMODE_CONTINOUS,
    Velocity := gvl.Axis_09_Jog_Velocity,
    Acceleration := 15,
    Deceleration := 20); // MC_Jog

// NETWORK 3
gvl.Axis_09_MC_Jog_Bw(
    Axis := GVL.Axis_09,
    JogBackwards := GVL.Axis_09_Jog_bw_Run,
    Mode := MC_JOGMODE_CONTINOUS,
    Velocity := gvl.Axis_09_Jog_Velocity,
    Acceleration := 15,
    Deceleration := 20); // MC_Jog

// NETWORK 4
GVL.Axis_09_MC_MoveAbsolute(
    Axis := GVL.Axis_09,
    Execute := GVL.Axis_09_MA_Enable_run,
    Position := gvl.Axis_09_Move_Val,
    Velocity := gvl.Axis_09_Velocity,
    Acceleration := gvl.Axis_09_accel,
    Deceleration := gvl.Axis_09_decel,
    Busy => GVL.Axis_09_Targeting); // MC_MoveAbsolute

// NETWORK 5
GVL.Axis_09_MC_MoveRelative(
    Axis := GVL.Axis_09,
    Execute := GVL.Axis_09_MR_Enable_run,
    Distance := gvl.Axis_09_Move_Val,
    Velocity := gvl.Axis_09_Velocity,
    Acceleration := gvl.Axis_09_accel,
    Deceleration := gvl.Axis_09_decel,
    Busy => GVL.Axis_09_Targeting); // MC_MoveRelative

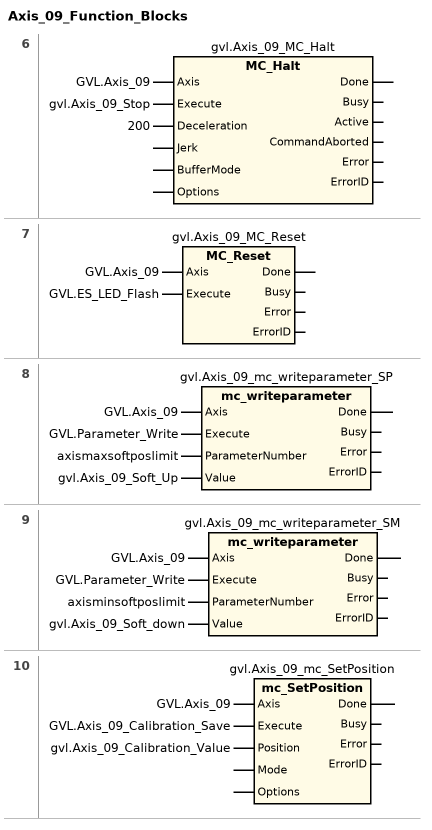
// NETWORK 6
gvl.Axis_09_MC_Halt(Axis := GVL.Axis_09, Execute := gvl.Axis_09_Stop, Deceleration := 200); // MC_Halt

// NETWORK 7
gvl.Axis_09_MC_Reset(Axis := GVL.Axis_09, Execute := GVL.ES_LED_Flash); // MC_Reset

// NETWORK 8
gvl.Axis_09_mc_writeparameter_SP(
    Axis := GVL.Axis_09,
    Execute := GVL.Parameter_Write,
    ParameterNumber := axismaxsoftposlimit,
    Value := gvl.Axis_09_Soft_Up); // mc_writeparameter

// NETWORK 9
gvl.Axis_09_mc_writeparameter_SM(
    Axis := GVL.Axis_09,
    Execute := GVL.Parameter_Write,
    ParameterNumber := axisminsoftposlimit,
    Value := gvl.Axis_09_Soft_down); // mc_writeparameter

// NETWORK 10
gvl.Axis_09_mc_SetPosition(
    Axis := GVL.Axis_09,
    Execute := GVL.Axis_09_Calibration_Save,
    Position := gvl.Axis_09_Calibration_Value); // mc_SetPosition

END_PROGRAM

// ---- POUs/Axis_09_Logic.TcPOU
PROGRAM Axis_09_Logic
VAR
	TON_0: TON;
	TON_1: TON;
	TON_2: TON;
	TON_3: TON;
	Axis_09_Velocity_Range: LREAL;
	Axis_09_Velocity_Scale: LREAL;
	Axis_09_Velocity_Raw: LREAL;
	Axis_09_Soft_Range: LREAL;
	Axis_09_Soft_Position: LREAL;
	Axis_09_Soft_Position_In_Range: LREAL;
END_VAR

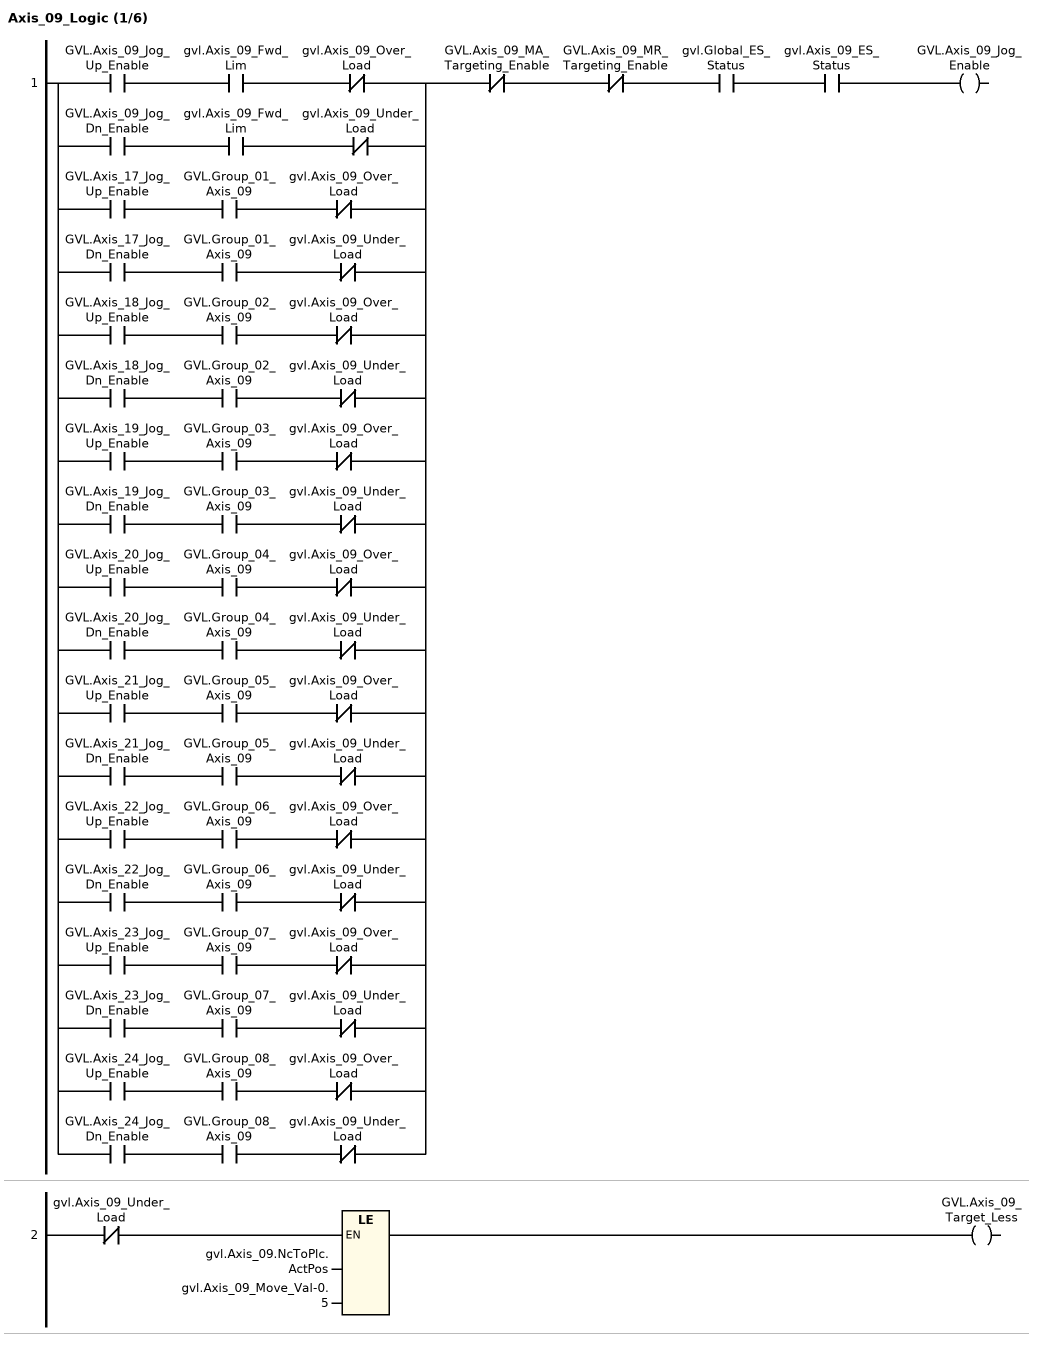
// NETWORK 1
GVL.Axis_09_Jog_Enable := (GVL.Axis_09_Jog_Up_Enable AND gvl.Axis_09_Fwd_Lim AND NOT gvl.Axis_09_Over_Load OR GVL.Axis_09_Jog_Dn_Enable AND gvl.Axis_09_Fwd_Lim AND NOT gvl.Axis_09_Under_Load OR GVL.Axis_17_Jog_Up_Enable AND GVL.Group_01_Axis_09 AND NOT gvl.Axis_09_Over_Load OR GVL.Axis_17_Jog_Dn_Enable AND GVL.Group_01_Axis_09 AND NOT gvl.Axis_09_Under_Load OR GVL.Axis_18_Jog_Up_Enable AND GVL.Group_02_Axis_09 AND NOT gvl.Axis_09_Over_Load OR GVL.Axis_18_Jog_Dn_Enable AND GVL.Group_02_Axis_09 AND NOT gvl.Axis_09_Under_Load OR GVL.Axis_19_Jog_Up_Enable AND GVL.Group_03_Axis_09 AND NOT gvl.Axis_09_Over_Load OR GVL.Axis_19_Jog_Dn_Enable AND GVL.Group_03_Axis_09 AND NOT gvl.Axis_09_Under_Load OR GVL.Axis_20_Jog_Up_Enable AND GVL.Group_04_Axis_09 AND NOT gvl.Axis_09_Over_Load OR GVL.Axis_20_Jog_Dn_Enable AND GVL.Group_04_Axis_09 AND NOT gvl.Axis_09_Under_Load OR GVL.Axis_21_Jog_Up_Enable AND GVL.Group_05_Axis_09 AND NOT gvl.Axis_09_Over_Load OR GVL.Axis_21_Jog_Dn_Enable AND GVL.Group_05_Axis_09 AND NOT gvl.Axis_09_Under_Load OR GVL.Axis_22_Jog_Up_Enable AND GVL.Group_06_Axis_09 AND NOT gvl.Axis_09_Over_Load OR GVL.Axis_22_Jog_Dn_Enable AND GVL.Group_06_Axis_09 AND NOT gvl.Axis_09_Under_Load OR GVL.Axis_23_Jog_Up_Enable AND GVL.Group_07_Axis_09 AND NOT gvl.Axis_09_Over_Load OR GVL.Axis_23_Jog_Dn_Enable AND GVL.Group_07_Axis_09 AND NOT gvl.Axis_09_Under_Load OR GVL.Axis_24_Jog_Up_Enable AND GVL.Group_08_Axis_09 AND NOT gvl.Axis_09_Over_Load OR GVL.Axis_24_Jog_Dn_Enable AND GVL.Group_08_Axis_09 AND NOT gvl.Axis_09_Under_Load) AND NOT GVL.Axis_09_MA_Targeting_Enable AND NOT GVL.Axis_09_MR_Targeting_Enable AND gvl.Global_ES_Status AND gvl.Axis_09_ES_Status;

// NETWORK 2
GVL.Axis_09_Target_Less := NOT gvl.Axis_09_Under_Load AND gvl.Axis_09.NcToPlc.ActPos <= (gvl.Axis_09_Move_Val-0.5);

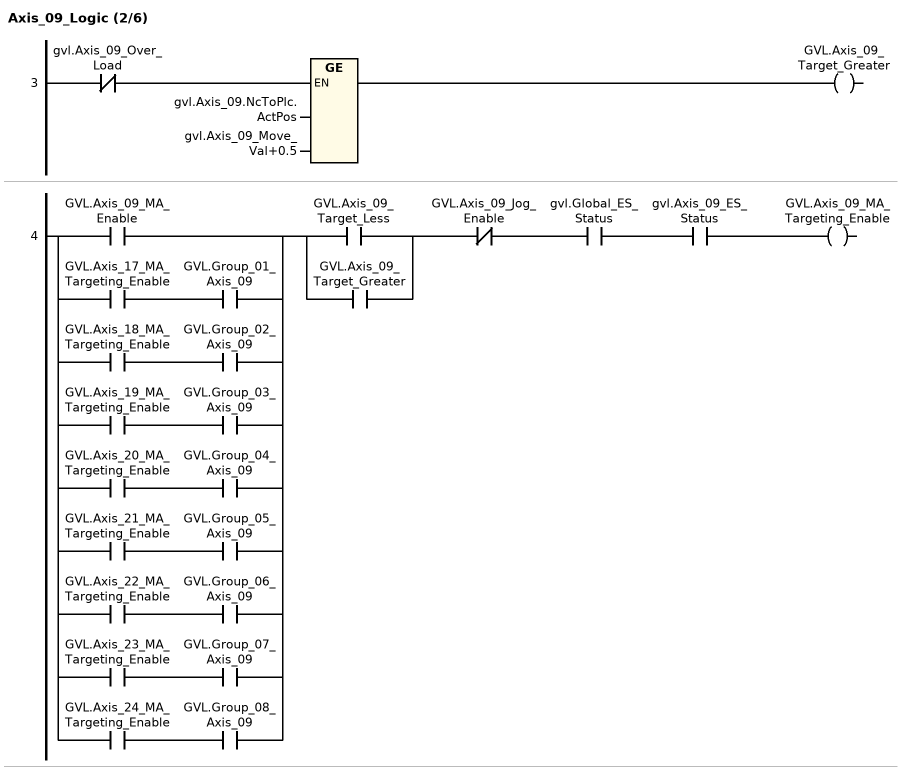
// NETWORK 3
GVL.Axis_09_Target_Greater := NOT gvl.Axis_09_Over_Load AND gvl.Axis_09.NcToPlc.ActPos >= (gvl.Axis_09_Move_Val+0.5);

// NETWORK 4
GVL.Axis_09_MA_Targeting_Enable := (GVL.Axis_09_MA_Enable OR GVL.Axis_17_MA_Targeting_Enable AND GVL.Group_01_Axis_09 OR GVL.Axis_18_MA_Targeting_Enable AND GVL.Group_02_Axis_09 OR GVL.Axis_19_MA_Targeting_Enable AND GVL.Group_03_Axis_09 OR GVL.Axis_20_MA_Targeting_Enable AND GVL.Group_04_Axis_09 OR GVL.Axis_21_MA_Targeting_Enable AND GVL.Group_05_Axis_09 OR GVL.Axis_22_MA_Targeting_Enable AND GVL.Group_06_Axis_09 OR GVL.Axis_23_MA_Targeting_Enable AND GVL.Group_07_Axis_09 OR GVL.Axis_24_MA_Targeting_Enable AND GVL.Group_08_Axis_09) AND (GVL.Axis_09_Target_Less OR GVL.Axis_09_Target_Greater) AND NOT GVL.Axis_09_Jog_Enable AND gvl.Global_ES_Status AND gvl.Axis_09_ES_Status;

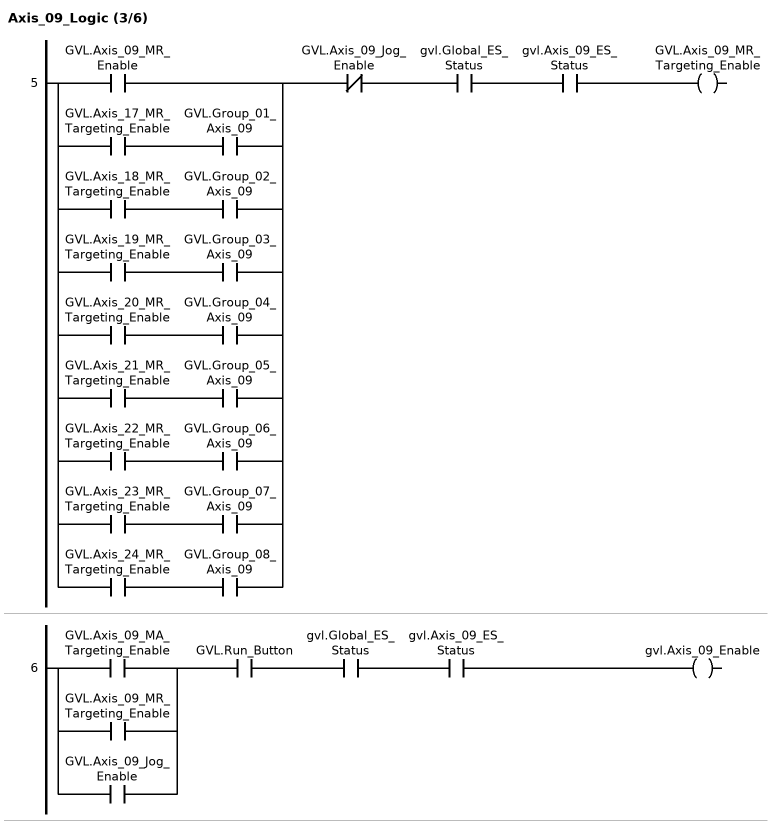
// NETWORK 5
GVL.Axis_09_MR_Targeting_Enable := (GVL.Axis_09_MR_Enable OR GVL.Axis_17_MR_Targeting_Enable AND GVL.Group_01_Axis_09 OR GVL.Axis_18_MR_Targeting_Enable AND GVL.Group_02_Axis_09 OR GVL.Axis_19_MR_Targeting_Enable AND GVL.Group_03_Axis_09 OR GVL.Axis_20_MR_Targeting_Enable AND GVL.Group_04_Axis_09 OR GVL.Axis_21_MR_Targeting_Enable AND GVL.Group_05_Axis_09 OR GVL.Axis_22_MR_Targeting_Enable AND GVL.Group_06_Axis_09 OR GVL.Axis_23_MR_Targeting_Enable AND GVL.Group_07_Axis_09 OR GVL.Axis_24_MR_Targeting_Enable AND GVL.Group_08_Axis_09) AND NOT GVL.Axis_09_Jog_Enable AND gvl.Global_ES_Status AND gvl.Axis_09_ES_Status;

// NETWORK 6
gvl.Axis_09_Enable := (GVL.Axis_09_MA_Targeting_Enable OR GVL.Axis_09_MR_Targeting_Enable OR GVL.Axis_09_Jog_Enable) AND GVL.Run_Button AND gvl.Global_ES_Status AND gvl.Axis_09_ES_Status;

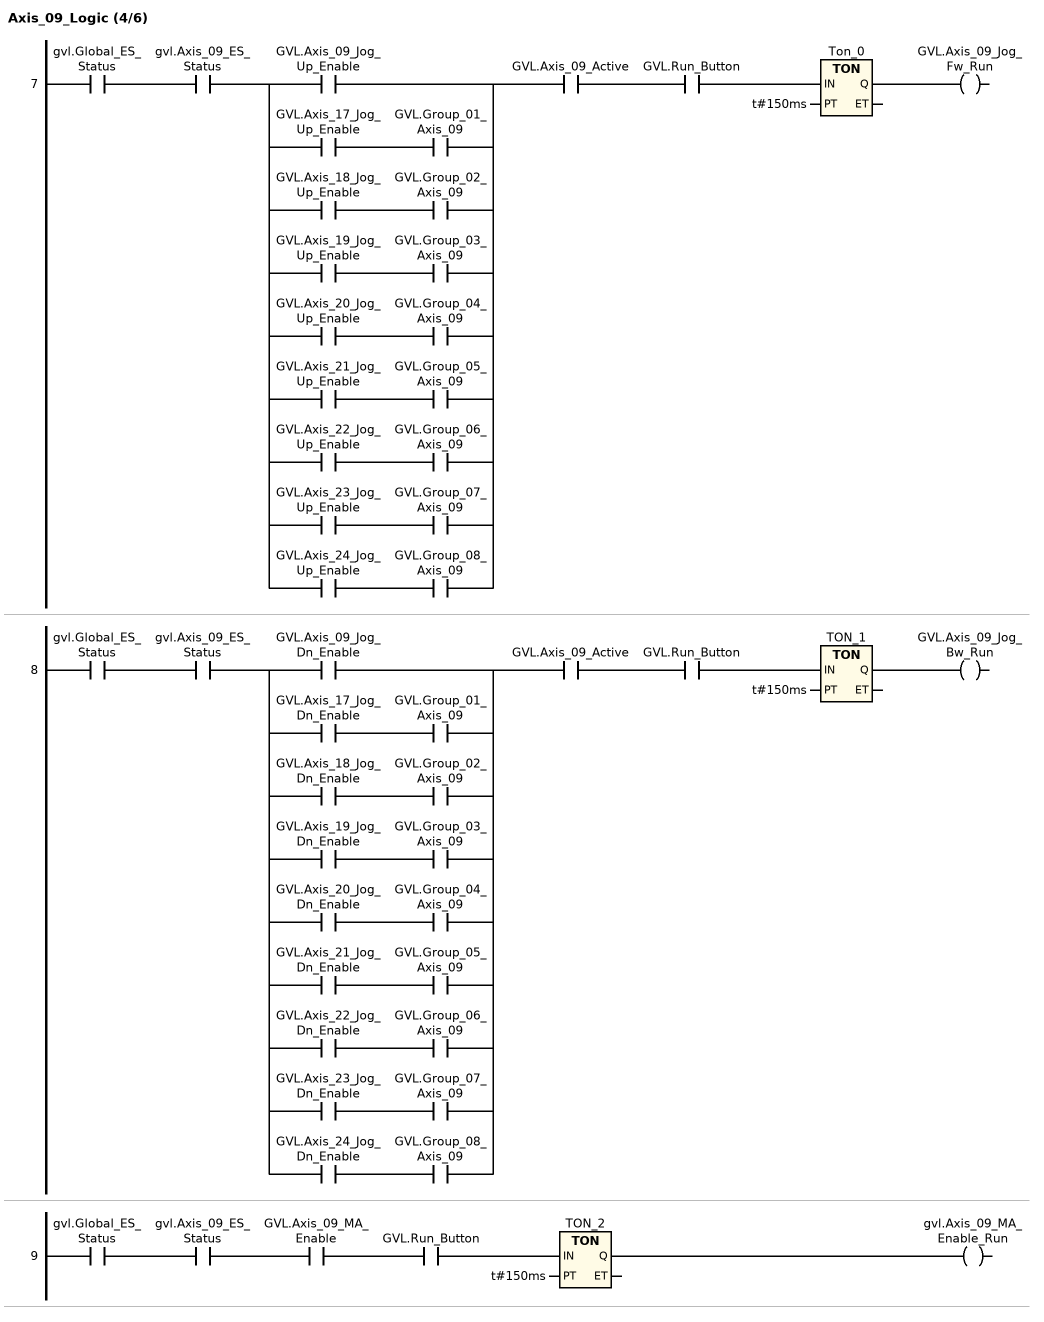
// NETWORK 7
Ton_0(IN := gvl.Global_ES_Status AND gvl.Axis_09_ES_Status AND (GVL.Axis_09_Jog_Up_Enable OR GVL.Axis_17_Jog_Up_Enable AND GVL.Group_01_Axis_09 OR GVL.Axis_18_Jog_Up_Enable AND GVL.Group_02_Axis_09 OR GVL.Axis_19_Jog_Up_Enable AND GVL.Group_03_Axis_09 OR GVL.Axis_20_Jog_Up_Enable AND GVL.Group_04_Axis_09 OR GVL.Axis_21_Jog_Up_Enable AND GVL.Group_05_Axis_09 OR GVL.Axis_22_Jog_Up_Enable AND GVL.Group_06_Axis_09 OR GVL.Axis_23_Jog_Up_Enable AND GVL.Group_07_Axis_09 OR GVL.Axis_24_Jog_Up_Enable AND GVL.Group_08_Axis_09) AND GVL.Axis_09_Active AND GVL.Run_Button, PT := t#150ms); // TON
GVL.Axis_09_Jog_Fw_Run := Ton_0.Q;

// NETWORK 8
TON_1(IN := gvl.Global_ES_Status AND gvl.Axis_09_ES_Status AND (GVL.Axis_09_Jog_Dn_Enable OR GVL.Axis_17_Jog_Dn_Enable AND GVL.Group_01_Axis_09 OR GVL.Axis_18_Jog_Dn_Enable AND GVL.Group_02_Axis_09 OR GVL.Axis_19_Jog_Dn_Enable AND GVL.Group_03_Axis_09 OR GVL.Axis_20_Jog_Dn_Enable AND GVL.Group_04_Axis_09 OR GVL.Axis_21_Jog_Dn_Enable AND GVL.Group_05_Axis_09 OR GVL.Axis_22_Jog_Dn_Enable AND GVL.Group_06_Axis_09 OR GVL.Axis_23_Jog_Dn_Enable AND GVL.Group_07_Axis_09 OR GVL.Axis_24_Jog_Dn_Enable AND GVL.Group_08_Axis_09) AND GVL.Axis_09_Active AND GVL.Run_Button, PT := t#150ms); // TON
GVL.Axis_09_Jog_Bw_Run := TON_1.Q;

// NETWORK 9
TON_2(IN := gvl.Global_ES_Status AND gvl.Axis_09_ES_Status AND GVL.Axis_09_MA_Enable AND GVL.Run_Button, PT := t#150ms); // TON
gvl.Axis_09_MA_Enable_Run := TON_2.Q;

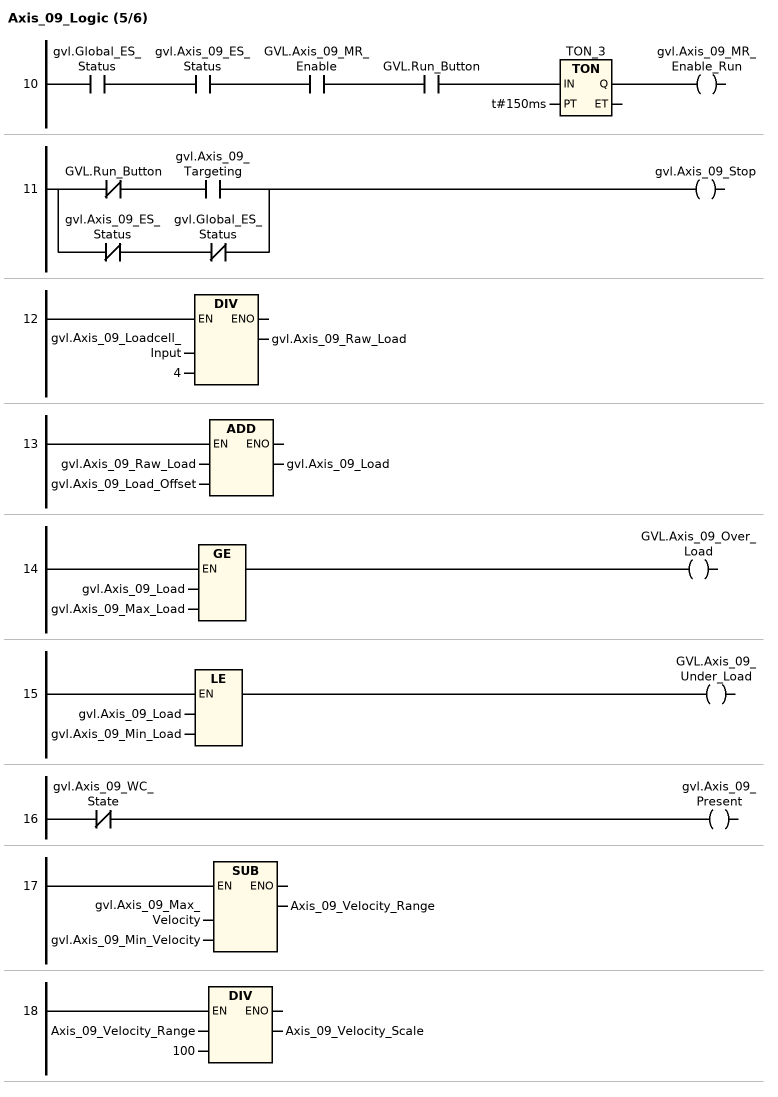
// NETWORK 10
TON_3(IN := gvl.Global_ES_Status AND gvl.Axis_09_ES_Status AND GVL.Axis_09_MR_Enable AND GVL.Run_Button, PT := t#150ms); // TON
gvl.Axis_09_MR_Enable_Run := TON_3.Q;

// NETWORK 11
gvl.Axis_09_Stop := NOT GVL.Run_Button AND gvl.Axis_09_Targeting OR NOT gvl.Axis_09_ES_Status AND NOT gvl.Global_ES_Status;

// NETWORK 12
gvl.Axis_09_Raw_Load := gvl.Axis_09_Loadcell_Input / 4;

// NETWORK 13
gvl.Axis_09_Load := gvl.Axis_09_Raw_Load + gvl.Axis_09_Load_Offset;

// NETWORK 14
GVL.Axis_09_Over_Load := gvl.Axis_09_Load >= gvl.Axis_09_Max_Load;

// NETWORK 15
GVL.Axis_09_Under_Load := gvl.Axis_09_Load <= gvl.Axis_09_Min_Load;

// NETWORK 16
gvl.Axis_09_Present := NOT gvl.Axis_09_WC_State;

// NETWORK 17
Axis_09_Velocity_Range := gvl.Axis_09_Max_Velocity - gvl.Axis_09_Min_Velocity;

// NETWORK 18
Axis_09_Velocity_Scale := Axis_09_Velocity_Range / 100;

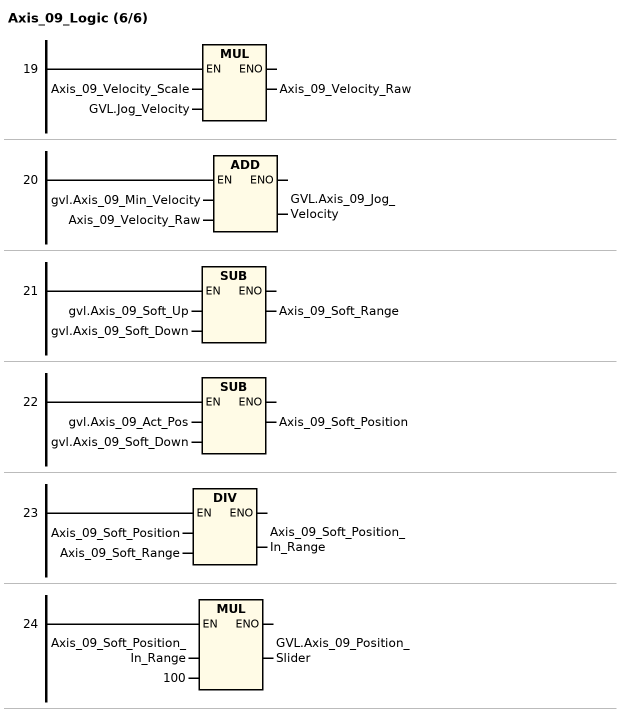
// NETWORK 19
Axis_09_Velocity_Raw := Axis_09_Velocity_Scale * GVL.Jog_Velocity;

// NETWORK 20
GVL.Axis_09_Jog_Velocity := gvl.Axis_09_Min_Velocity + Axis_09_Velocity_Raw;

// NETWORK 21
Axis_09_Soft_Range := gvl.Axis_09_Soft_Up - gvl.Axis_09_Soft_Down;

// NETWORK 22
Axis_09_Soft_Position := gvl.Axis_09_Act_Pos - gvl.Axis_09_Soft_Down;

// NETWORK 23
Axis_09_Soft_Position_In_Range := Axis_09_Soft_Position / Axis_09_Soft_Range;

// NETWORK 24
GVL.Axis_09_Position_Slider := Axis_09_Soft_Position_In_Range * 100;

END_PROGRAM

// ---- POUs/Axis_10_Function_Blocks.TcPOU
PROGRAM Axis_10_Function_Blocks
VAR
END_VAR

